FUNCTION_BLOCK E_REND
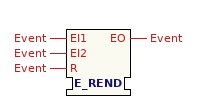
  EVENT_INPUT
    EI1;
    EI2;
    R;
  END_EVENT
  EVENT_OUTPUT
    EO;
  END_EVENT
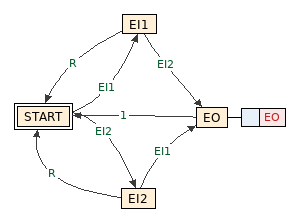
  EC_STATES
    START;
    EI1;
    EO : -> EO;
    EI2;
  END_STATES
  EC_TRANSITIONS
    START TO EI2 := EI2;
    START TO EI1 := EI1;
    EI2 TO START := R;
    EI1 TO START := R;
    EI1 TO EO := EI2;
    EI2 TO EO := EI1;
    EO TO START := 1;
  END_TRANSITIONS
END_FUNCTION_BLOCK
